FUNCTION CheckLRangeSigned : LINT
VAR_INPUT
	value, lower, upper: LINT;
END_VAR

{noflow}

IF (value < lower) THEN
	CheckLRangeSigned := lower;
	oaksGVL.udiCheckLRangeSigned := oaksGVL.udiCheckLRangeSigned + 1;
ELSIF(value > upper) THEN
	CheckLRangeSigned := upper;
	oaksGVL.udiCheckLRangeSigned := oaksGVL.udiCheckLRangeSigned + 1;
ELSE
	CheckLRangeSigned := value;
END_IF

{flow}

END_FUNCTION

(* stored: Version 1.1.0.1, ProductVersion 3.1.4022.18
   POU CheckLRangeSigned: Id {5c53c7dd-d3d1-4218-99b2-5eb7555f04e6}, SpecialFunc CheckLRangeSigned *)
